GLOBALCONSTANTS DefaultPool_Joystick (* Global constants *)
  PACKAGE Uebungen::const::UT::Joystick;
  VAR_GLOBAL CONSTANT
    ISO_DESIGNATOR_WIDTH : UINT := 80;
    ISO_DESIGNATOR_HEIGHT : UINT := 80;
    ISO_MASK_SIZE : UINT := 480;
    ISO_VERSION_LABEL : STRING;
    MASK_WIDTH : UINT := 480;
    MASK_HEIGHT : UINT := 480;
    WorkingSet : UINT := 0;
    DataMask : UINT := 1000;
    Container_3000 : UINT := 3000;
    Container_3001 : UINT := 3001;
    Container_3002 : UINT := 3002;
    Container_3003 : UINT := 3003;
    OutputString_WS : UINT := 11500;
    DM_main : UINT := 20000;
    I1 : UINT := 20001;
    I2 : UINT := 20002;
    I3 : UINT := 20003;
    I4 : UINT := 20004;
    FontAttributes_WS : UINT := 23500;
    AuxInput2_32000 : UINT := 32000;
    AuxInput2_32001 : UINT := 32001;
    AuxInput2_32002 : UINT := 32002;
    AuxInput2_32003 : UINT := 32003;
    AuxObjectPointer_33000 : UINT := 33000;
    AuxObjectPointer_33001 : UINT := 33001;
    AuxObjectPointer_33002 : UINT := 33002;
    AuxObjectPointer_33003 : UINT := 33003;
    AuxObjectPointer_33004 : UINT := 33004;
    AuxObjectPointer_33005 : UINT := 33005;
    AuxObjectPointer_33006 : UINT := 33006;
    AuxObjectPointer_33007 : UINT := 33007;
    AuxObjectPointer_33008 : UINT := 33008;
    AuxObjectPointer_33009 : UINT := 33009;
    AuxObjectPointer_33010 : UINT := 33010;
    AuxObjectPointer_33011 : UINT := 33011;
    AuxObjectPointer_33012 : UINT := 33012;
    AuxObjectPointer_33013 : UINT := 33013;
    AuxObjectPointer_33014 : UINT := 33014;
    AuxObjectPointer_33015 : UINT := 33015;
  END_VAR
END_GLOBALCONSTANTS
